FUNCTION_BLOCK LowpassFilter
VAR_INPUT
	r_Input : REAL;
	r_Tao : REAL;
END_VAR
VAR_OUTPUT
	r_Output : REAL;
END_VAR
VAR
	r_Output_k1 : REAL;
	r_Time : REAL := 0.01;
END_VAR

r_Output := (r_Input + (r_Input*r_Tao/r_Time))/(1+r_Tao/r_Time);
r_Output_k1 := r_Output;

END_FUNCTION_BLOCK

(* stored: Version 1.1.0.1, ProductVersion 3.1.4022.12
   POU LowpassFilter: Id {3c208087-fc2a-4825-b1f0-f09fa7e5ce23}, SpecialFunc None *)
